// TIA Portal V17 export
// export: Created 2021-12-03T08:14:55.5709821Z, ExportSetting WithDefaults, DisplayName Totally Integrated Automation Portal, DisplayVersion V17, DisplayName TIA Portal Openness, DisplayVersion V17, DisplayName TIA Portal Version Control Interface, DisplayVersion V17, DisplayName STEP 7 Professional, DisplayVersion V17, DisplayName STEP 7 Safety, DisplayVersion V17, DisplayName WinCC Advanced, DisplayVersion V17
TYPE "UDT_TRACE"
// stored: IsFailsafeCompliant false
   STRUCT
      state : Array[0..10] of Int;
      event : Array[0..10] of Int;
      action : Array[0..10] of Int;
   END_STRUCT;
END_TYPE
